PROGRAM Control_SFC
VAR
	iSetManual: BOOL;
	iSetAuto: BOOL;
	iAutoStart: BOOL;
	iManualLeft: BOOL;
	iManualRight: BOOL;
	iAutoStop: BOOL;
	iStop: BOOL;
	
	xMode: STRING;
	xAutomatic: BOOL;
	xManual: BOOL;
	xAutoStart: BOOL;
	xAutoStop: BOOL;
	xManualLeft: BOOL;
	xManualRight: BOOL;
END_VAR

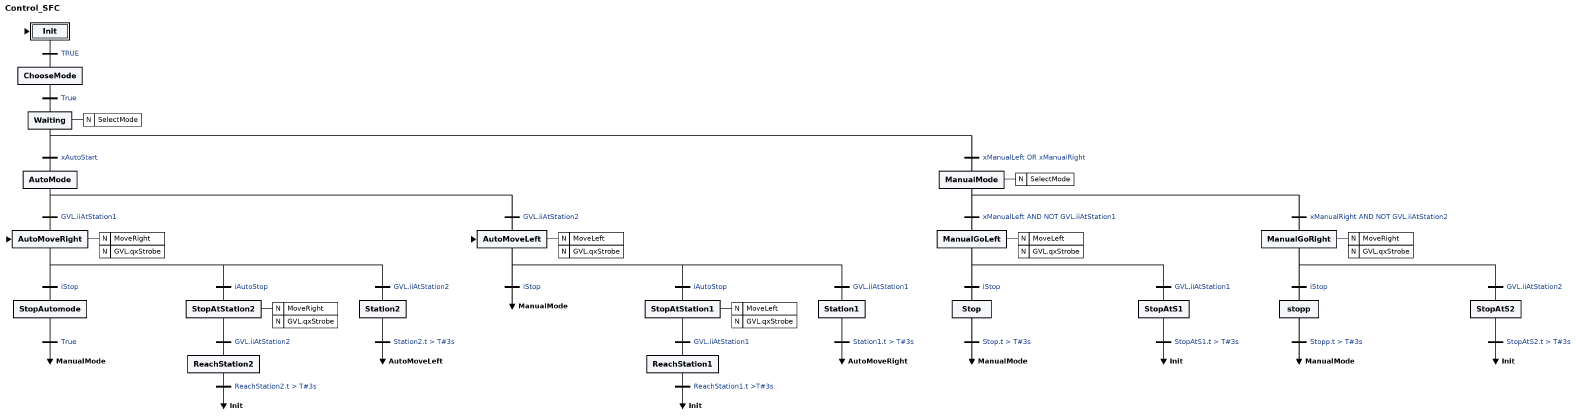
INITIAL_STEP Init:
END_STEP
TRANSITION FROM Init TO ChooseMode
    := TRUE;
END_TRANSITION
STEP ChooseMode:
END_STEP
TRANSITION FROM ChooseMode TO Waiting
    := True;
END_TRANSITION
STEP Waiting:
    SelectMode(N);
END_STEP
TRANSITION FROM Waiting TO AutoMode
    := xAutoStart;
END_TRANSITION
STEP AutoMode:
END_STEP
TRANSITION FROM AutoMode TO AutoMoveRight
    := GVL.iiAtStation1;
END_TRANSITION
STEP AutoMoveRight:
    MoveRight(N);
    GVL.qxStrobe(N);
END_STEP
TRANSITION FROM AutoMoveRight TO StopAutomode
    := iStop;
END_TRANSITION
STEP StopAutomode:
END_STEP
TRANSITION FROM StopAutomode TO ManualMode
    := True;
END_TRANSITION
TRANSITION FROM AutoMoveRight TO StopAtStation2
    := iAutoStop;
END_TRANSITION
TRANSITION FROM AutoMoveRight TO Station2
    := GVL.iiAtStation2;
END_TRANSITION
STEP Station2:
END_STEP
TRANSITION FROM Station2 TO AutoMoveLeft
    := Station2.t > T#3s;
END_TRANSITION
STEP StopAtStation2:
    MoveRight(N);
    GVL.qxStrobe(N);
END_STEP
TRANSITION FROM StopAtStation2 TO ReachStation2
    := GVL.iiAtStation2;
END_TRANSITION
STEP ReachStation2:
END_STEP
TRANSITION FROM ReachStation2 TO Init
    := ReachStation2.t > T#3s;
END_TRANSITION
TRANSITION FROM AutoMode TO AutoMoveLeft
    := GVL.iiAtStation2;
END_TRANSITION
STEP AutoMoveLeft:
    MoveLeft(N);
    GVL.qxStrobe(N);
END_STEP
TRANSITION FROM AutoMoveLeft TO ManualMode
    := iStop;
END_TRANSITION
TRANSITION FROM AutoMoveLeft TO StopAtStation1
    := iAutoStop;
END_TRANSITION
TRANSITION FROM AutoMoveLeft TO Station1
    := GVL.iiAtStation1;
END_TRANSITION
STEP Station1:
END_STEP
TRANSITION FROM Station1 TO AutoMoveRight
    := Station1.t > T#3s;
END_TRANSITION
STEP StopAtStation1:
    MoveLeft(N);
    GVL.qxStrobe(N);
END_STEP
TRANSITION FROM StopAtStation1 TO ReachStation1
    := GVL.iiAtStation1;
END_TRANSITION
STEP ReachStation1:
END_STEP
TRANSITION FROM ReachStation1 TO Init
    := ReachStation1.t >T#3s;
END_TRANSITION
TRANSITION FROM Waiting TO _ManualMode
    := xManualLeft OR xManualRight;
END_TRANSITION
STEP _ManualMode:  // name as stored:  ManualMode
    SelectMode(N);
END_STEP
TRANSITION FROM _ManualMode TO ManualGoLeft
    := xManualLeft AND NOT GVL.iiAtStation1;
END_TRANSITION
STEP ManualGoLeft:
    MoveLeft(N);
    GVL.qxStrobe(N);
END_STEP
TRANSITION FROM ManualGoLeft TO Stop
    := iStop;
END_TRANSITION
STEP Stop:
END_STEP
TRANSITION FROM Stop TO ManualMode
    := Stop.t > T#3s;
END_TRANSITION
TRANSITION FROM ManualGoLeft TO StopAtS1
    := GVL.iiAtStation1;
END_TRANSITION
STEP StopAtS1:
END_STEP
TRANSITION FROM StopAtS1 TO Init
    := StopAtS1.t > T#3s;
END_TRANSITION
TRANSITION FROM _ManualMode TO ManualGoRight
    := xManualRight AND NOT GVL.iiAtStation2;
END_TRANSITION
STEP ManualGoRight:
    MoveRight(N);
    GVL.qxStrobe(N);
END_STEP
TRANSITION FROM ManualGoRight TO stopp
    := iStop;
END_TRANSITION
STEP stopp:
END_STEP
TRANSITION FROM stopp TO ManualMode
    := Stopp.t > T#3s;
END_TRANSITION
TRANSITION FROM ManualGoRight TO StopAtS2
    := GVL.iiAtStation2;
END_TRANSITION
STEP StopAtS2:
END_STEP
TRANSITION FROM StopAtS2 TO Init
    := StopAtS2.t > T#3s;
END_TRANSITION

ACTION MoveLeft:
GVL.qxDir := -1;
END_ACTION

ACTION MoveRight:
GVL.qxDir := 1;
END_ACTION

ACTION SelectMode:
xAutoStart := FALSE;
xAutoStop := FALSE;
xManualLeft := FALSE;
xManualRight := FALSE;

IF iSetManual THEN
	xAutomatic := FALSE;
	xManual := TRUE;
	xMode := 'Manual';
ELSIF iSetAuto THEN 
	xAutomatic := TRUE;
	xManual := FALSE;
	xMode := 'Automatic';
END_IF

IF xAutomatic THEN
	IF iAutoStart THEN
		xAutoStart := TRUE;
		xAutoStop := FALSE;
	ELSIF iAutoStop THEN
		xAutoStart := FALSE;
		xAutoStop := TRUE;
	END_IF
END_IF

IF xManual THEN
	IF iManualLeft THEN
		xManualLeft := TRUE;
		xManualRight := FALSE;
	ELSIF iManualRight THEN
		xManualLeft := FALSE;
		xManualRight := TRUE;
	END_IF
END_IF
END_ACTION

END_PROGRAM

(* stored: Version 1.1.0.1, ProductVersion 3.1.4024.12
   POU Control_SFC: Id {ebbfde16-cde5-43c6-ac76-0869aa22951e}, SpecialFunc None
   Action MoveLeft: Id {8c290c3f-536c-4c88-a812-832b8f97d928}
   Action MoveRight: Id {b0f02329-c1b3-487d-9d16-2d354bd5d1e0}
   Action SelectMode: Id {8885e23e-1e8c-4dcb-9a5d-0ad1cb2f817d} *)
